FUNCTION_BLOCK SymbolProvider_1
VAR_INPUT
END_VAR
VAR_OUTPUT
END_VAR
VAR
	symbolReader		: FB_JsonReadWriteDatatype;
END_VAR


METHOD GetDatatype : T_MaxString
VAR_INPUT
	symbol			: ANY;
END_VAR

GetDatatype := symbolReader.GetDatatypeNameByAddress(pData := symbol.pValue, nData := TO_UDINT(symbol.diSize));
END_METHOD


METHOD GetFullName : T_MaxString
VAR_INPUT
	symbol			: ANY;
END_VAR

GetFullName := symbolReader.GetSymbolNameByAddress(pData := symbol.pValue, nData := TO_UDINT(symbol.diSize));
END_METHOD


(* Returns full symbol name without its GVL or PRG name at the beginning
	example: for symbol 'MAIN.bStart' returns 'bStart'
*)
METHOD GetNameWithoutGlobalNameSpace : T_MaxString
VAR_INPUT
	symbol			: ANY;
END_VAR

GetNameWithoutGlobalNameSpace := symbolReader.GetSymbolNameByAddress(pData := symbol.pValue, nData := TO_UDINT(symbol.diSize));
GetNameWithoutGlobalNameSpace := RIGHT(STR := GetNameWithoutGlobalNameSpace, SIZE := LEN(GetNameWithoutGlobalNameSpace) - FIND(STR1 := GetNameWithoutGlobalNameSpace, STR2 := '.'));
END_METHOD

END_FUNCTION_BLOCK

(* stored: Version 1.1.0.1, ProductVersion 3.1.4024.11
   POU SymbolProvider_1: Id {3eb6e77d-d059-4a6e-a91a-7b1db2f1c35b}, SpecialFunc None
   Method GetDatatype: Id {c228097f-b18b-47e0-a983-684b1bbad4b7}
   Method GetFullName: Id {634b3c22-dbca-443a-9cee-c3e15c0203fc}
   Method GetNameWithoutGlobalNameSpace: Id {08b39e72-ae31-4cdc-a9c5-5dd70c689f80} *)
